TYPE MyStructureExtended EXTENDS MyStructure :
STRUCT
    member2     : UDINT;            //          Another property
END_STRUCT
END_TYPE

(* stored: Version 1.1.0.1, ProductVersion 3.1.4024.11
   DUT MyStructureExtended: Id {9f7fa53e-2b51-4a26-9680-c182cabee752} *)
